{region '#Template'}
	{attribute 'Version' := '5.0.0.0'}
	{attribute 'Tags' := '"LCID": "1031", "Text": "RA, HC, Building, Energy"'}
	{attribute 'Tags' := '"LCID": "1033", "Text": "RA, HC, Building, Energy"'}
	{attribute 'Using' := '"Type": "Template", "URI": "Site"'}
	{attribute 'Description' := '"LCID": "1031", "Text": "Gebäude Energieniveau"'}
	{attribute 'Description' := '"LCID": "1033", "Text": "Building energy level"'}
{endregion}
FUNCTION_BLOCK FB_BA_BuildingEnergyLevel EXTENDS FB_BA_View

VAR_INPUT CONSTANT
	EnergLvlMan						: FB_BA_MV_Op ;     
	EnergLvlPr						: FB_BA_MV_Op;      
	Sched							: FB_BA_SchedM;
END_VAR

VAR	                            		
	DeMuxEnergLvl					: FB_BA_DMUX_B08;
	DeMuxSched						: FB_BA_DMUX_B04;
	PrioSwi							: FB_BA_PrioSwi_UDI08;
END_VAR

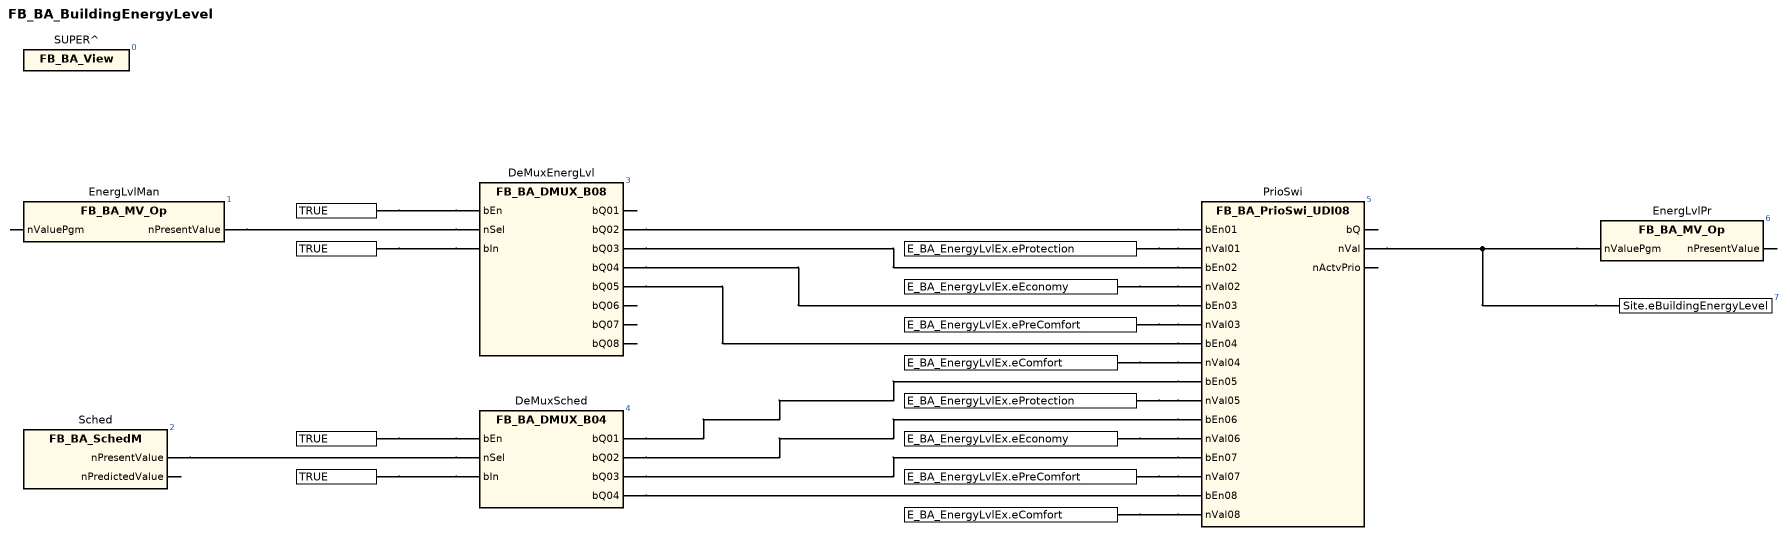
SUPER^(); // FB_BA_View
EnergLvlMan(); // FB_BA_MV_Op
Sched(); // FB_BA_SchedM
DeMuxEnergLvl(bEn := TRUE, nSel := EnergLvlMan.nPresentValue, bIn := TRUE); // FB_BA_DMUX_B08
DeMuxSched(bEn := TRUE, nSel := Sched.nPresentValue, bIn := TRUE); // FB_BA_DMUX_B04
PrioSwi(
    bEn01 := DeMuxEnergLvl.bQ02,
    nVal01 := E_BA_EnergyLvlEx.eProtection,
    bEn02 := DeMuxEnergLvl.bQ03,
    nVal02 := E_BA_EnergyLvlEx.eEconomy,
    bEn03 := DeMuxEnergLvl.bQ04,
    nVal03 := E_BA_EnergyLvlEx.ePreComfort,
    bEn04 := DeMuxEnergLvl.bQ05,
    nVal04 := E_BA_EnergyLvlEx.eComfort,
    bEn05 := DeMuxSched.bQ01,
    nVal05 := E_BA_EnergyLvlEx.eProtection,
    bEn06 := DeMuxSched.bQ02,
    nVal06 := E_BA_EnergyLvlEx.eEconomy,
    bEn07 := DeMuxSched.bQ03,
    nVal07 := E_BA_EnergyLvlEx.ePreComfort,
    bEn08 := DeMuxSched.bQ04,
    nVal08 := E_BA_EnergyLvlEx.eComfort); // FB_BA_PrioSwi_UDI08
EnergLvlPr(nValuePgm := PrioSwi.nVal); // FB_BA_MV_Op
Site.eBuildingEnergyLevel := PrioSwi.nVal;

METHOD FB_init : BOOL
VAR_INPUT
	bInitRetains : BOOL; // if TRUE; the retain variables are initialized (warm start / cold start)
	bInCopyCode : BOOL;  // if TRUE; the instance afterwards gets moved into the copy code (online change)
END_VAR
EnergLvlMan.iParent			:= THIS^;	
EnergLvlMan.iLabel			:= LblCtl_BuildingEnergyLevelManual;
EnergLvlMan.aStateText[1]	:= txtEvent_Auto;
EnergLvlMan.aStateText[2]	:= txtEvent_Protection;
EnergLvlMan.aStateText[3]	:= txtEvent_Economy;
EnergLvlMan.aStateText[4]	:= txtEvent_PreComfort;
EnergLvlMan.aStateText[5]	:= txtEvent_Comfort;
EnergLvlMan.nValueRm		:= 1;

EnergLvlPr.iParent			:= THIS^;	
EnergLvlPr.iLabel			:= LblCtl_BuildingEnergyLevelActual;
EnergLvlPr.aStateText[1]	:= txtEvent_Protection;
EnergLvlPr.aStateText[2]	:= txtEvent_Economy;
EnergLvlPr.aStateText[3]	:= txtEvent_PreComfort;
EnergLvlPr.aStateText[4]	:= txtEvent_Comfort;
EnergLvlPr.nValueRm			:= 1;
											
Sched.iParent				:= THIS^;	
Sched.iLabel				:= LblCtl_BuildingEnergyLevelSched; 
Sched.aStateText[1]			:= txtEvent_Protection;
Sched.aStateText[2]			:= txtEvent_Economy;
Sched.aStateText[3]			:= txtEvent_PreComfort;
Sched.aStateText[4]			:= txtEvent_Comfort;
Sched.nPredictTime			:= 0;


Sched.aWeek		:= F_BA_SchedWeekly3xM(E_BA_WeekDay.eMonday, E_BA_WeekDay.eFriday, T#0H, E_BA_EnergyLvlEx.eProtection, T#6H, E_BA_EnergyLvlEx.eComfort, T#20H, E_BA_EnergyLvlEx.eProtection);
(* alternatively
Sched.nDefaultValue										:= E_BA_EnergyLvlEx.eProtection;
Sched.bWriteWeekly										:= FALSE;
//	Monday
Sched.aWeek[E_BA_Weekday.eMonday,1].eState				:= E_BA_SchedEntryState.eValue;
Sched.aWeek[E_BA_Weekday.eMonday,1].uValue.udiVal		:= E_BA_EnergyLvlEx.eComfort;
Sched.aWeek[E_BA_Weekday.eMonday,1].stTime.nHour		:= 6;
Sched.aWeek[E_BA_Weekday.eMonday,1].stTime.nMinute		:= 0;
Sched.aWeek[E_BA_Weekday.eMonday,1].stTime.nSecond		:= 0;
Sched.aWeek[E_BA_Weekday.eMonday,2].eState				:= E_BA_SchedEntryState.eValue;
Sched.aWeek[E_BA_Weekday.eMonday,2].uValue.udiVal		:= E_BA_EnergyLvlEx.eEconomy;
Sched.aWeek[E_BA_Weekday.eMonday,2].stTime.nHour		:= 20;
Sched.aWeek[E_BA_Weekday.eMonday,2].stTime.nMinute		:= 0;
Sched.aWeek[E_BA_Weekday.eMonday,2].stTime.nSecond		:= 0;
Sched.aWeek[E_BA_Weekday.eMonday,3].eState				:= E_BA_SchedEntryState.eValue;
Sched.aWeek[E_BA_Weekday.eMonday,3].uValue.udiVal		:= E_BA_EnergyLvlEx.eProtection;
Sched.aWeek[E_BA_Weekday.eMonday,3].stTime.nHour		:= 0;
Sched.aWeek[E_BA_Weekday.eMonday,3].stTime.nMinute		:= 0;
Sched.aWeek[E_BA_Weekday.eMonday,3].stTime.nSecond		:= 0;
//	Tuesday
Sched.aWeek[E_BA_Weekday.eTuesday,1].eState				:= E_BA_SchedEntryState.eValue;
Sched.aWeek[E_BA_Weekday.eTuesday,1].uValue.udiVal		:= E_BA_EnergyLvlEx.eComfort;
Sched.aWeek[E_BA_Weekday.eTuesday,1].stTime.nHour		:= 6;
Sched.aWeek[E_BA_Weekday.eTuesday,1].stTime.nMinute		:= 0;
Sched.aWeek[E_BA_Weekday.eTuesday,1].stTime.nSecond		:= 0;
Sched.aWeek[E_BA_Weekday.eTuesday,2].eState				:= E_BA_SchedEntryState.eValue;
Sched.aWeek[E_BA_Weekday.eTuesday,2].uValue.udiVal		:= E_BA_EnergyLvlEx.eEconomy;
Sched.aWeek[E_BA_Weekday.eTuesday,2].stTime.nHour		:= 20;
Sched.aWeek[E_BA_Weekday.eTuesday,2].stTime.nMinute		:= 0;
Sched.aWeek[E_BA_Weekday.eTuesday,2].stTime.nSecond		:= 0;
Sched.aWeek[E_BA_Weekday.eTuesday,3].eState				:= E_BA_SchedEntryState.eValue;
Sched.aWeek[E_BA_Weekday.eTuesday,3].uValue.udiVal		:= E_BA_EnergyLvlEx.eProtection;
Sched.aWeek[E_BA_Weekday.eTuesday,3].stTime.nHour		:= 0;
Sched.aWeek[E_BA_Weekday.eTuesday,3].stTime.nMinute		:= 0;
Sched.aWeek[E_BA_Weekday.eTuesday,3].stTime.nSecond		:= 0;
//	Wednesday
Sched.aWeek[E_BA_Weekday.eWednesday,1].eState			:= E_BA_SchedEntryState.eValue;
Sched.aWeek[E_BA_Weekday.eWednesday,1].uValue.udiVal	:= E_BA_EnergyLvlEx.eComfort;
Sched.aWeek[E_BA_Weekday.eWednesday,1].stTime.nHour		:= 6;
Sched.aWeek[E_BA_Weekday.eWednesday,1].stTime.nMinute	:= 0;
Sched.aWeek[E_BA_Weekday.eWednesday,1].stTime.nSecond	:= 0;
Sched.aWeek[E_BA_Weekday.eWednesday,2].eState			:= E_BA_SchedEntryState.eValue;
Sched.aWeek[E_BA_Weekday.eWednesday,2].uValue.udiVal	:= E_BA_EnergyLvlEx.eEconomy;
Sched.aWeek[E_BA_Weekday.eWednesday,2].stTime.nHour		:= 20;
Sched.aWeek[E_BA_Weekday.eWednesday,2].stTime.nMinute	:= 0;
Sched.aWeek[E_BA_Weekday.eWednesday,2].stTime.nSecond	:= 0;
Sched.aWeek[E_BA_Weekday.eWednesday,3].eState			:= E_BA_SchedEntryState.eValue;
Sched.aWeek[E_BA_Weekday.eWednesday,3].uValue.udiVal	:= E_BA_EnergyLvlEx.eProtection;
Sched.aWeek[E_BA_Weekday.eWednesday,3].stTime.nHour		:= 0;
Sched.aWeek[E_BA_Weekday.eWednesday,3].stTime.nMinute	:= 0;
Sched.aWeek[E_BA_Weekday.eWednesday,3].stTime.nSecond	:= 0;
//	Thursday
Sched.aWeek[E_BA_Weekday.eThursday,1].eState			:= E_BA_SchedEntryState.eValue;
Sched.aWeek[E_BA_Weekday.eThursday,1].uValue.udiVal		:=E_BA_EnergyLvlEx.eComfort;
Sched.aWeek[E_BA_Weekday.eThursday,1].stTime.nHour		:= 6;
Sched.aWeek[E_BA_Weekday.eThursday,1].stTime.nMinute	:= 0;
Sched.aWeek[E_BA_Weekday.eThursday,1].stTime.nSecond	:= 0;
Sched.aWeek[E_BA_Weekday.eThursday,2].eState			:= E_BA_SchedEntryState.eValue;
Sched.aWeek[E_BA_Weekday.eThursday,2].uValue.udiVal		:= E_BA_EnergyLvlEx.eEconomy;
Sched.aWeek[E_BA_Weekday.eThursday,2].stTime.nHour		:= 20;
Sched.aWeek[E_BA_Weekday.eThursday,2].stTime.nMinute	:= 0;
Sched.aWeek[E_BA_Weekday.eThursday,2].stTime.nSecond	:= 0;
Sched.aWeek[E_BA_Weekday.eThursday,3].eState			:= E_BA_SchedEntryState.eValue;
Sched.aWeek[E_BA_Weekday.eThursday,3].uValue.udiVal		:= E_BA_EnergyLvlEx.eProtection;
Sched.aWeek[E_BA_Weekday.eThursday,3].stTime.nHour		:= 0;
Sched.aWeek[E_BA_Weekday.eThursday,3].stTime.nMinute	:= 0;
Sched.aWeek[E_BA_Weekday.eThursday,3].stTime.nSecond	:= 0;
//	Friday
Sched.aWeek[E_BA_Weekday.eFriday,1].eState				:= E_BA_SchedEntryState.eValue;
Sched.aWeek[E_BA_Weekday.eFriday,1].uValue.udiVal		:= E_BA_EnergyLvlEx.eComfort;
Sched.aWeek[E_BA_Weekday.eFriday,1].stTime.nHour		:= 6;
Sched.aWeek[E_BA_Weekday.eFriday,1].stTime.nMinute		:= 0;
Sched.aWeek[E_BA_Weekday.eFriday,1].stTime.nSecond		:= 0;
Sched.aWeek[E_BA_Weekday.eFriday,2].eState				:= E_BA_SchedEntryState.eValue;
Sched.aWeek[E_BA_Weekday.eFriday,2].uValue.udiVal		:= E_BA_EnergyLvlEx.eEconomy;
Sched.aWeek[E_BA_Weekday.eFriday,2].stTime.nHour		:= 20;
Sched.aWeek[E_BA_Weekday.eFriday,2].stTime.nMinute		:= 0;
Sched.aWeek[E_BA_Weekday.eFriday,2].stTime.nSecond		:= 0;
Sched.aWeek[E_BA_Weekday.eFriday,3].eState				:= E_BA_SchedEntryState.eValue;
Sched.aWeek[E_BA_Weekday.eFriday,3].uValue.udiVal		:= E_BA_EnergyLvlEx.eProtection;
Sched.aWeek[E_BA_Weekday.eFriday,3].stTime.nHour		:= 0;
Sched.aWeek[E_BA_Weekday.eFriday,3].stTime.nMinute		:= 0;
Sched.aWeek[E_BA_Weekday.eFriday,3].stTime.nSecond		:= 0;

*)
END_METHOD

END_FUNCTION_BLOCK

(* stored: Version 1.1.0.1, ProductVersion 3.1.4024.12
   POU FB_BA_BuildingEnergyLevel: Id {c9580724-b208-4b56-8e3a-5f10802513d1}, SpecialFunc None
   Method FB_init: Id {c9a734f6-2016-4655-a682-8a3ea58c17b4} *)
